Yaskawa INFORM job: OK_R2_O54(90,90)AWOK.JBI

/JOB
//NAME OK_R2_O54(90,90)AWOK
///FOLDERNAME X4
//POS
///NPOS 78,78,78,4,0,0
///TOOL 0
///POSTYPE PULSE
///PULSE
C00000=-93051,-79362,-65205,778,51067,-80227
C00001=-102340,-35835,-41511,5626,59216,-83768
C00002=-125546,16839,18753,3325,112791,-78678
C00003=-125193,10566,16887,3408,110705,-78608
C00004=-125338,4752,11778,3355,110867,-78656
C00005=-125339,5428,13792,3329,109979,-78685
C00006=-125338,4752,11778,3355,110867,-78656
C00007=-125193,10566,16887,3408,110705,-78608
C00008=-115080,14427,23905,-7535,109251,-79269
C00009=-115024,12462,22117,-7526,109345,-79255
C00010=-115080,14427,23905,-7535,109251,-79269
C00011=-115005,11939,18951,-7603,111013,-79358
C00012=-114782,18324,21018,-7636,113026,-79408
C00013=-113825,18538,21218,-7247,113101,-79052
C00014=-124914,16975,20215,-1386,107196,80319
C00015=-124236,11021,16275,-1169,106579,80567
C00016=-122697,11964,18588,2367,106235,80981
C00017=-120670,5046,12163,-39,106065,81841
C00018=-120671,5702,14099,-39,105210,81841
C00019=-120670,5046,12163,-39,106065,81841
C00020=-120669,10918,17333,-38,105901,81841
C00021=-120664,13367,22956,-36,103700,81844
C00022=-120664,11809,21544,-36,103769,81844
C00023=-120664,13367,22956,-36,103700,81844
C00024=-122037,10946,17358,-470,105896,81356
C00025=-139789,-6887,-4826,16075,98624,73872
C00026=-138229,-38529,-21283,19349,54466,73206
C00027=-138229,-40865,-27841,18734,57153,73708
C00028=-132021,-97421,-62751,-309,78611,78036
C00029=-120704,-95876,-65781,-23,90169,81849
C00030=-120673,-21168,-25487,-19,103760,81857
C00031=-120653,18427,20993,-37,117310,81846
C00032=-120655,11367,17955,-38,115552,81845
C00033=-121497,-11331,-6525,860,109222,81413
C00034=-121497,-10892,-5008,855,108515,81408
C00035=-121497,-11331,-6525,860,109222,81413
C00036=-120655,11367,17955,-38,115552,81845
C00037=-120694,13185,22347,-55,113782,81831
C00038=-120694,11662,20968,-55,113850,81831
C00039=-120694,13185,22347,-55,113782,81831
C00040=-120653,18427,20993,-37,117310,81846
C00041=-120651,11571,12338,-39,115316,81848
C00042=-120667,-12436,-9975,5103,110550,-80129
C00043=-135504,-6240,-6756,236,112251,-85585
C00044=-137190,-7292,-5881,-325,111171,-86209
C00045=-120667,-10291,-8310,5106,110627,-80126
C00046=-120668,-12803,-11522,5133,111310,-80096
C00047=-121617,-10867,-8882,24199,110654,-59852
C00048=-120947,-10739,-8748,24393,110442,-59629
C00049=-122195,-10499,-10079,24194,111672,-59860
C00050=-120668,-12296,-9868,24722,110258,-59302
C00051=-120673,-21168,-25487,-19,103760,81857
C00052=-120704,-95876,-65781,-23,90169,81849
C00053=-130855,-87373,-58995,-278,81466,78422
C00054=-136695,-120484,-67139,5650,47887,75110
C00055=-137539,-56218,-39498,4931,63890,75574
C00056=-131681,-19905,-16777,-233,89960,78120
C00057=-120669,-12962,-10380,28389,117609,62624
C00058=-120672,-9547,-7734,28423,117721,62655
C00059=-117379,-11083,-8859,29637,116491,63761
C00060=-120669,-10818,-8721,28411,117680,62644
C00061=-120669,-13330,-11926,28606,118283,62815
C00062=-129485,-33603,-26883,33888,106061,67003
C00063=-125777,-38657,-27628,40061,99870,69835
C00064=-126781,-39737,-31772,40200,101880,70163
C00065=-143129,-24300,-21495,37253,110498,66038
C00066=-121196,-24675,-20129,124,101317,78289
C00067=-120667,-12839,-10285,-5181,110528,79304
C00068=-117483,-12687,-10169,-4149,110720,81268
C00069=-117385,-11098,-8764,-4116,110675,81308
C00070=-120668,-13212,-11835,-5211,111288,80066
C00071=-120668,-10700,-8629,-5184,110608,80097
C00072=-121676,-11141,-9212,-23754,110128,60210
C00073=-120670,-9866,-7984,-24814,110314,59255
C00074=-117642,-12567,-12784,-24203,112644,59957
C00075=-120669,-12924,-10350,-24793,110209,59279
C00076=-120669,-12924,-10350,-24793,110209,59279
C00077=11166,-12924,-10350,-24793,47970,59279
BC00000=116331,719030,247437
BC00001=116331,719030,247437
BC00002=96614,768022,366028
BC00003=96614,768022,366028
BC00004=96614,768022,366028
BC00005=96614,768022,366028
BC00006=96614,768022,366028
BC00007=96614,768022,366028
BC00008=96614,768022,366028
BC00009=96615,768022,366026
BC00010=96614,768022,366028
BC00011=96614,768022,366028
BC00012=96614,768022,366028
BC00013=96614,768022,366028
BC00014=185541,760110,383191
BC00015=185541,760110,383191
BC00016=185541,760110,383191
BC00017=185541,760110,383191
BC00018=185541,760110,383191
BC00019=185541,760110,383191
BC00020=185541,760110,383191
BC00021=185541,760110,383191
BC00022=185541,760110,383191
BC00023=185541,760110,383191
BC00024=185541,760110,383191
BC00025=185541,760110,383191
BC00026=185541,760110,383191
BC00027=186496,695562,383191
BC00028=185541,760110,383191
BC00029=335238,776240,348735
BC00030=335238,776240,348735
BC00031=335238,776240,348735
BC00032=335238,776240,348735
BC00033=335238,776240,348735
BC00034=335238,776240,348735
BC00035=335238,776240,348735
BC00036=335238,776240,348735
BC00037=335238,776240,348735
BC00038=335238,776240,348735
BC00039=335238,776240,348735
BC00040=335238,776240,348735
BC00041=335238,776240,348735
BC00042=285998,785762,347557
BC00043=286869,778873,323533
BC00044=286958,778172,321088
BC00045=286959,778172,321094
BC00046=286959,778172,321094
BC00047=333658,775324,288502
BC00048=333658,775324,288502
BC00049=333658,775324,288502
BC00050=327859,781535,309861
BC00051=335238,776240,348735
BC00052=335238,776240,348735
BC00053=185541,760110,383191
BC00054=185541,760110,383191
BC00055=185541,760110,383191
BC00056=185541,760110,383191
BC00057=95166,795746,300724
BC00058=95853,790325,281822
BC00059=96128,788157,274258
BC00060=96127,788156,274261
BC00061=96127,788156,274261
BC00062=197341,788073,274067
BC00063=197397,787973,273924
BC00064=197397,787973,273924
BC00065=197397,787973,273924
BC00066=154600,786173,335680
BC00067=146285,785823,347678
BC00068=145583,780411,328767
BC00069=145352,778625,322540
BC00070=145302,778243,321207
BC00071=145302,778243,321207
BC00072=106462,775188,290679
BC00073=105705,776740,294751
BC00074=110279,781194,310283
BC00075=110279,758211,310283
BC00076=110279,666768,310283
BC00077=110279,666768,310283
EC00000=798156,556475
EC00001=798156,556475
EC00002=798156,556475
EC00003=798156,556475
EC00004=798156,556475
EC00005=798156,556475
EC00006=798156,556475
EC00007=798156,556475
EC00008=798156,556475
EC00009=798155,556475
EC00010=798156,556475
EC00011=798156,556475
EC00012=798156,556475
EC00013=798156,556475
EC00014=798156,556475
EC00015=798156,556475
EC00016=798156,556475
EC00017=798156,556475
EC00018=798156,556475
EC00019=798156,556475
EC00020=798156,556475
EC00021=798156,556475
EC00022=798156,556475
EC00023=798156,556475
EC00024=798156,556475
EC00025=798156,556475
EC00026=798156,556475
EC00027=798156,556475
EC00028=798156,556475
EC00029=798156,556475
EC00030=798156,556475
EC00031=798156,556475
EC00032=798156,556475
EC00033=798156,556475
EC00034=798156,556475
EC00035=798156,556475
EC00036=798156,556475
EC00037=798156,556475
EC00038=798156,556475
EC00039=798156,556475
EC00040=798156,556475
EC00041=798156,556475
EC00042=798156,556475
EC00043=798153,556474
EC00044=798153,556474
EC00045=798156,556475
EC00046=798156,556475
EC00047=798156,556475
EC00048=798156,556475
EC00049=798156,556475
EC00050=798156,556475
EC00051=798156,556475
EC00052=798156,556475
EC00053=798156,556475
EC00054=798156,556475
EC00055=798156,556475
EC00056=798156,556475
EC00057=798156,556475
EC00058=798156,556475
EC00059=798154,556474
EC00060=798156,556475
EC00061=798156,556475
EC00062=798156,556475
EC00063=798156,556475
EC00064=798156,556475
EC00065=798156,556475
EC00066=798156,556475
EC00067=798156,556475
EC00068=798156,556475
EC00069=798156,556475
EC00070=798156,556475
EC00071=798156,556475
EC00072=798156,556475
EC00073=798156,556475
EC00074=798156,556475
EC00075=798156,556475
EC00076=798156,556475
EC00077=798156,556475
///POSTYPE BASE
///RECTAN
///RCONF 0,0,0,0,0,0,0,0,0,0,0,0,0,0,0,0,0,0,0,0,0,0,0,0
P00006=0.222,-3.123,-1.508,0.0000,0.0000,0.0000
P00021=-0.225,-6.128,-0.405,0.0000,0.0000,0.0000
P00022=0.222,-3.123,-1.508,0.0000,0.0000,0.0000
P00023=0.143,-0.036,0.682,0.0000,0.0000,0.0000
//INST
///DATE 2024/04/13 16:49
///ATTR SC,RW
///GROUP1 RB1,BS1
///GROUP2 ST1
NOP
'OK_r2_O54(90,90)
'Path S1566
SFTOF3D
MOVJ C00000 BC00000 VJ=100.00  +MOVJ EC00000 VJ=100.00
MOVJ C00001 BC00001 VJ=100.00  +MOVJ EC00001 VJ=100.00
MOVJ C00002 BC00002 VJ=100.00  +MOVJ EC00002 VJ=100.00
MOVL C00003 BC00003 V=400.0  +MOVJ EC00003 VJ=100.00
SMOVL C00004 BC00004 V=100.0  +MOVJ EC00004
SREFP 3 C00005 BC00005  +REFP EC00005
CALL JOB:SEARCH-R1-S13D
SET P022 P006
SFTON3D P022
SMOVL C00006 BC00006 V=100.0  +MOVJ EC00006
SMOVL C00007 BC00007 V=166.7  +MOVJ EC00007
SMOVL C00008 BC00008 V=100.0  +MOVJ EC00008
SREFP 3 C00009 BC00009  +REFP EC00009
CALL JOB:SEARCH-R1-S13D
SET P022 P006
SFTON3D P022
SMOVL C00010 BC00010 V=100.0  +MOVJ EC00010
SMOVL C00011 BC00011 V=166.7  +MOVJ EC00011
MOVL C00012 BC00012 V=1000.0  +MOVJ EC00012 VJ=100.00
MOVJ C00013 BC00013 VJ=100.00  +MOVJ EC00013 VJ=99.00
'Path S1567
SFTOF3D
MOVJ C00014 BC00014 VJ=100.00  +MOVJ EC00014 VJ=100.00
MOVL C00015 BC00015 V=400.0  +MOVJ EC00015 VJ=100.00
SMOVL C00016 BC00016 V=100.0  +MOVJ EC00016
SMOVL C00017 BC00017 V=50.0  +MOVJ EC00017
SREFP 3 C00018 BC00018  +REFP EC00018
CALL JOB:SEARCH-R1-S13D
SET P023 P006
SFTON3D P023
SMOVL C00019 BC00019 V=60.0  +MOVJ EC00019
SMOVL C00020 BC00020 V=100.0  +MOVJ EC00020
SMOVL C00021 BC00021 V=166.7  +MOVJ EC00021
SREFP 3 C00022 BC00022  +REFP EC00022
CALL JOB:SEARCH-R1-S13D
SET P023 P006
SFTON3D P023
SMOVL C00023 BC00023 V=100.0  +MOVJ EC00023
SMOVL C00024 BC00024 V=100.0  +MOVJ EC00024
MOVL C00025 BC00025 V=166.7  +MOVJ EC00025 VJ=100.00
MOVJ C00026 BC00026 VJ=100.00  +MOVJ EC00026 VJ=100.00
MOVJ C00027 BC00027 VJ=100.00  +MOVJ EC00027 VJ=50.00
MOVJ C00028 BC00028 VJ=100.00  +MOVJ EC00028 VJ=100.00
MOVJ C00029 BC00029 VJ=100.00  +MOVJ EC00029 VJ=100.00
MOVJ C00030 BC00030 VJ=15.00  +MOVJ EC00030 VJ=100.00
'Path S1568
SFTOF3D
MOVJ C00031 BC00031 VJ=100.00  +MOVJ EC00031 VJ=100.00
MOVL C00032 BC00032 V=333.3  +MOVJ EC00032 VJ=100.00
SMOVL C00033 BC00033 V=100.0  +MOVJ EC00033
SREFP 3 C00034 BC00034  +REFP EC00034
CALL JOB:SEARCH-R1-S13D
SET P021 P006
SFTON3D P021
SMOVL C00035 BC00035 V=100.0  +MOVJ EC00035
SMOVL C00036 BC00036 V=250.0  +MOVJ EC00036
SMOVL C00037 BC00037 V=100.0  +MOVJ EC00037
SREFP 3 C00038 BC00038  +REFP EC00038
CALL JOB:SEARCH-R1-S13D
SET P021 P006
SFTON3D P021
SMOVL C00039 BC00039 V=100.0  +MOVJ EC00039
MOVL C00040 BC00040 V=1000.0  +MOVJ EC00040 VJ=100.00
MOVJ C00041 BC00041 VJ=100.00  +MOVJ EC00041 VJ=10.00
'Path W1569
SFTOF3D
SFTON3D P021
MOVJ C00042 BC00042 VJ=100.00  +MOVJ EC00042 VJ=100.00
MOVJ C00043 BC00043 VJ=100.00  +MOVJ EC00043 VJ=100.00
SMOVL C00044 BC00044 V=100.0 PL=0  +MOVJ EC00044
SREFP 1 C00045 BC00045  +REFP EC00045
SREFP 2 C00046 BC00046  +REFP EC00046
MACRO1 MJ#(0) ARGF14
ARCON
SMOVL C00047 BC00047 V=10.0  +MOVJ EC00047
SMOVL C00048 BC00048 V=10.0  +MOVJ EC00048
ARCOF
SMOVL C00049 BC00049 V=400.0  +MOVJ EC00049
SMOVL C00050 BC00050 V=1000.0  +MOVJ EC00050
SFTOF3D
MOVJ C00051 BC00051 VJ=100.00  +MOVJ EC00051 VJ=100.00
MOVJ C00052 BC00052 VJ=50.00  +MOVJ EC00052 VJ=100.00
MOVJ C00053 BC00053 VJ=100.00  +MOVJ EC00053 VJ=100.00
MOVJ C00054 BC00054 VJ=100.00  +MOVJ EC00054 VJ=50.00
MOVJ C00055 BC00055 VJ=50.00  +MOVJ EC00055 VJ=50.00
MOVJ C00056 BC00056 VJ=25.00  +MOVJ EC00056 VJ=100.00
SFTOF3D
'Path W1570
SFTOF3D
SFTON3D P023
MOVJ C00057 BC00057 VJ=100.00  +MOVJ EC00057 VJ=100.00
SMOVL C00058 BC00058 V=333.3  +MOVJ EC00058
SMOVL C00059 BC00059 V=166.7 PL=0  +MOVJ EC00059
SREFP 1 C00060 BC00060  +REFP EC00060
SREFP 2 C00061 BC00061  +REFP EC00061
MACRO1 MJ#(0) ARGF14
ARCON
SMOVL C00062 BC00062 V=10.0  +MOVJ EC00062
SMOVL C00063 BC00063 V=10.0  +MOVJ EC00063
ARCOF
SMOVL C00064 BC00064 V=400.0  +MOVJ EC00064
SMOVL C00065 BC00065 V=416.7  +MOVJ EC00065
SFTOF3D
MOVJ C00066 BC00066 VJ=100.00  +MOVJ EC00066 VJ=50.00
'Path W1571
SFTOF3D
SFTON3D P022
MOVJ C00067 BC00067 VJ=100.00  +MOVJ EC00067 VJ=100.00
MOVJ C00068 BC00068 VJ=100.00  +MOVJ EC00068 VJ=100.00
SMOVL C00069 BC00069 V=100.0 PL=0  +MOVJ EC00069
SREFP 1 C00070 BC00070  +REFP EC00070
SREFP 2 C00071 BC00071  +REFP EC00071
MACRO1 MJ#(0) ARGF14
ARCON
SMOVL C00072 BC00072 V=10.0  +MOVJ EC00072
ARCOF
SMOVL C00073 BC00073 V=400.0  +MOVJ EC00073
SMOVL C00074 BC00074 V=1000.0  +MOVJ EC00074
SFTOF3D
MOVJ C00075 BC00075 VJ=100.00  +MOVJ EC00075 VJ=100.00
MOVJ C00076 BC00076 VJ=100.00  +MOVJ EC00076 VJ=100.00
MOVJ C00077 BC00077 VJ=70.00  +MOVJ EC00077 VJ=100.00
END
